TYPE "Ergebnisdaten"
TITLE = Datentyp mit den Ergebnisdaten
VERSION : 0.1
//HIer werden die zu sendenen Ergebnisdaten definiert
   STRUCT
      one : Bool;   // beschreibung one
      two : Byte;   // beschreibung two
      three : Word;   // beschreibung three
      four : DWord;   // beschreibung four
      five : LWord;   // beschreibung five
      six : SInt;   // beschreibung six
      seven : USInt;   // beschreibung seven
      eight : Int;   // beschreibung eight
      nine : UInt;   // beschreibung nine
      ten : DInt;   // beschreibung ten
      eleven : UDInt;   // beschreibung eleven
      twelve : LInt;   // beschreibung twelve
      thirteen : ULInt;   // beschreibung thirteen
      fourteen : Real;   // beschreibung fourteen
      fifteen : LReal;   // beschreibung fifteen
      sixteen : Char;   // beschreibung sixteen
      seventeen : WChar;   // beschreibung seventeen
      eighteen : String;   // beschreibung eighteen
      nineteen : WString;   // beschreibung nineteen
      twenty {InstructionName := 'DTL'; LibVersion := '1.0'} : DTL;   // beschreibung twenty
      twentyone : Array[0..10] of Byte;   // beschreibung twentyone
      twentytwo : Struct   // beschreibung twentytwo
         one : Bool;   // twentytwo one
         two : Int;   // twentytwo two
         three : DInt;   // twentytwo three
      END_STRUCT;
      twentythree : "Status";   // beschreibung twentythree
   END_STRUCT;

END_TYPE

